FUNCTION_BLOCK ASSEMBLE_AW_FROM_AB (* this Function combines the 2 AB (BYTE) adapters to a AW (WORD) *)
  (* Standard: 61499-2; Description: Copyright (c) 2026 Meisterschulen am Ostbahnhof SPDX-License-Identifier: EPL-2.0 *)
  (* Version 1.0, 2026-05-16, Franz Höpfinger, Meisterschulen am Ostbahnhof, initial API and implementation and/or initial documentation *)
  PACKAGE adapter::assembling;
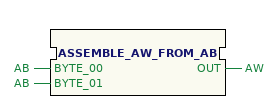
  SOCKETS
    BYTE_00 : adapter::types::unidirectional::AB; (* Byte 0 *)
    BYTE_01 : adapter::types::unidirectional::AB; (* Byte 1 *)
  END_SOCKETS
  PLUGS
    OUT : adapter::types::unidirectional::AW; (* WORD Output *)
  END_PLUGS
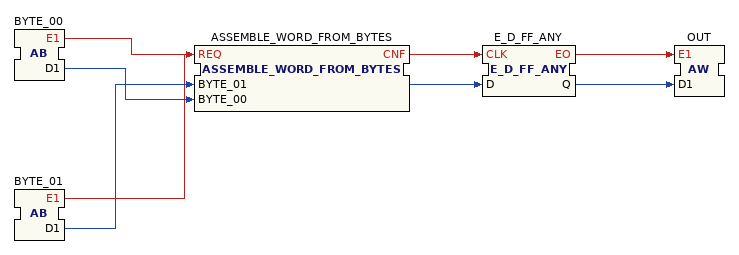
  FBS
    ASSEMBLE_WORD_FROM_BYTES : eclipse4diac::utils::assembling::ASSEMBLE_WORD_FROM_BYTES;
    E_D_FF_ANY : iec61499::events::E_D_FF_ANY;
  END_FBS
  EVENT_CONNECTIONS
    BYTE_00.E1 TO ASSEMBLE_WORD_FROM_BYTES.REQ;
    BYTE_01.E1 TO ASSEMBLE_WORD_FROM_BYTES.REQ;
    ASSEMBLE_WORD_FROM_BYTES.CNF TO E_D_FF_ANY.CLK;
    E_D_FF_ANY.EO TO OUT.E1;
  END_CONNECTIONS
  DATA_CONNECTIONS
    ASSEMBLE_WORD_FROM_BYTES. TO E_D_FF_ANY.D;
    E_D_FF_ANY.Q TO OUT.D1;
    BYTE_01.D1 TO ASSEMBLE_WORD_FROM_BYTES.BYTE_01;
    BYTE_00.D1 TO ASSEMBLE_WORD_FROM_BYTES.BYTE_00;
  END_CONNECTIONS
END_FUNCTION_BLOCK
